// TIA Portal project "TIA_ControlTankSystem_VCSimit" (V16)

(* hardware
DEVICE "S71500/ET200MP station_1"  S7-1500 station
   slot 0: "Rail_0"  Rack  6ES7 590-1***0-0AA0
   slot 1: "PLC_1"  CPU 1511-1 PN  6ES7 511-1AK01-0AB0  V2.6
      slot 3: "CPU display_1"  6ES7591-1AA00-0AA0
      slot 32768: "PROFINET interface_1"  X1
         slot 32769: "Port_1"  X1 P1
         slot 32770: "Port_2"  X1 P2
DEVICE "S71500/ET200MP station_2"  S7-1500 station
   slot 0: "Rail_0"  Rack  6ES7 590-1***0-0AA0
   slot 1: "PLC_2"  CPU 1511-1 PN  6ES7 511-1AK01-0AB0  V2.8
      slot 3: "CPU display_1"  6ES7591-1AA00-0AA0
      slot 32768: "PROFINET interface_1"  X1
         slot 32769: "Port_1"  X1 P1
         slot 32770: "Port_2"  X1 P2
      slot 34817: "Virtual CP interface port_1"  Virtual CP interface port  Virtual CP interface port
DEVICE "ET 200SP station_1"  ET 200SP-Station
   slot 0: "Rack_0"  Rack  6ES5 710-8MAx1
   slot 0: "IO device_1"  IM 155-6 PN HF  6ES7 155-6AU00-0CN0  V4.2
   slot 1: "DI 8x24VDC HF_1"  DI 8x24VDC HF  6ES7 131-6BF00-0CA0  V2.0
      slot 1: "DI 8x24VDC HF_1"  DI 8x24VDC HF
   slot 2: "DI 8x24VDC HF_2"  DI 8x24VDC HF  6ES7 131-6BF00-0CA0  V2.0
      slot 1: "DI 8x24VDC HF_2"  DI 8x24VDC HF
   slot 3: "DI 8x24VDC HF_3"  DI 8x24VDC HF  6ES7 131-6BF00-0CA0  V2.0
      slot 1: "DI 8x24VDC HF_3"  DI 8x24VDC HF
   slot 4: "DQ 8x24VDC/0.5A HF_1"  DQ 8x24VDC/0.5A HF  6ES7 132-6BF00-0CA0  V2.0
      slot 1: "DQ 8x24VDC/0.5A HF_1"  DQ 8x24VDC/0.5A HF
   slot 5: "DQ 8x24VDC/0.5A HF_2"  DQ 8x24VDC/0.5A HF  6ES7 132-6BF00-0CA0  V2.0
      slot 1: "DQ 8x24VDC/0.5A HF_2"  DQ 8x24VDC/0.5A HF
   slot 6: "AI 2xU/I 2-,4-wire HS_1"  AI 2xU/I 2-,4-wire HS  6ES7 134-6HB00-0DA1  V2.0
      slot 1: "AI 2xU/I 2-,4-wire HS_1"  AI 2xU/I 2-,4-wire HS
   slot 7: "AI 2xU/I 2-,4-wire HS_2"  AI 2xU/I 2-,4-wire HS  6ES7 134-6HB00-0DA1  V2.0
      slot 1: "AI 2xU/I 2-,4-wire HS_2"  AI 2xU/I 2-,4-wire HS
   slot 8: "AI 2xU/I 2-,4-wire HS_3"  AI 2xU/I 2-,4-wire HS  6ES7 134-6HB00-0DA1  V2.0
      slot 1: "AI 2xU/I 2-,4-wire HS_3"  AI 2xU/I 2-,4-wire HS
   slot 9: "AQ 2xU/I HS_1"  AQ 2xU/I HS  6ES7 135-6HB00-0DA1  V2.0
      slot 1: "AQ 2xU/I HS_1"  AQ 2xU/I HS
   slot 10: "AQ 2xU/I HS_2"  AQ 2xU/I HS  6ES7 135-6HB00-0DA1  V2.0
      slot 1: "AQ 2xU/I HS_2"  AQ 2xU/I HS
   slot 11: "Server module_1"  Server module  6ES7 193-6PA00-0AA0  V1.1
      slot 1: "Server module_1"  Server module
   slot 127: "BA 2xRJ45"  BA 2xRJ45  6ES7 193-6AR00-0AA0  V0.0
      slot 1: "Port_1"  X1 P1 R  6ES7 193-6AR00-0AA0  V0.0
      slot 2: "Port_2"  X1 P2 R  6ES7 193-6AR00-0AA0  V0.0
DEVICE "PC-System_1"  SIMATIC PC station
   slot 0: "SIMATIC PC station"  Rail  SIMATIC PC-Station  V1.0
      slot 125: "Stationmanager"  Station_Manager  V6.0.4
   slot 1: "HMI_RT_1"  WinCC RT Advanced  6AV2 104-0xxxx-xxxx  16.0.0.0
      slot 33792: "Computer interface"  Host interface
   slot 2: "IE general_1"  IE General  IE_CP  V8.2.0
*)

// ===== PLC "PLC_1"  CPU 1511-1 PN =====

VAR_GLOBAL   // PLC tag table "Default tag table"
   "Motor2_SpeedRaw" AT %MW0 : Int;
   "Motor2_Speed" AT %MD2 : Real;
   "Tank2_Level" AT %MD6 : Real;
   "Tank2_LevelRaw" AT %MW10 : Int;
   "Motor2_SpeedSPRaw" AT %MW12 : Int;
   "Motor2_SpeedSP" AT %MD14 : Real;
   "Motor2_VFDCMD" AT %M18.0 : Bool;
END_VAR

DATA_BLOCK "ReadBuffer"   // DB2
{ S7_Optimized_Access := 'FALSE' }
VERSION : 0.1
   VAR
      Speed_2 : Int;
      BoolStatus_2 : Word;
      Level_2 : Int;
   END_VAR
BEGIN
END_DATA_BLOCK

DATA_BLOCK "ModbusConfig"   // DB3
{ S7_Optimized_Access := 'TRUE' }
VERSION : 0.1
   VAR
      ReadConfig : TCON_IP_v4;
      WriteConfig : TCON_IP_v4;
   END_VAR
BEGIN
   ReadConfig.InterfaceId := 64;
   ReadConfig.ID := 30;
   ReadConfig.ActiveEstablished := true;
   ReadConfig.RemoteAddress.ADDR[1] := 192;
   ReadConfig.RemoteAddress.ADDR[2] := 168;
   ReadConfig.RemoteAddress.ADDR[3] := 0;
   ReadConfig.RemoteAddress.ADDR[4] := 12;
   ReadConfig.RemotePort := 502;
   ReadConfig.ConnectionType := 11;
   WriteConfig.InterfaceId := 64;
   WriteConfig.ID := 31;
   WriteConfig.ConnectionType := 11;
   WriteConfig.ActiveEstablished := true;
   WriteConfig.RemoteAddress.ADDR[1] := 192;
   WriteConfig.RemoteAddress.ADDR[2] := 168;
   WriteConfig.RemoteAddress.ADDR[3] := 0;
   WriteConfig.RemoteAddress.ADDR[4] := 12;
   WriteConfig.RemotePort := 502;
END_DATA_BLOCK

DATA_BLOCK "WriteBuffer"   // DB4
{ S7_Optimized_Access := 'FALSE' }
VERSION : 0.1
   VAR
      SpeedSP_2 : Int;
      BoolStatus_2 : Int;
   END_VAR
BEGIN
END_DATA_BLOCK

DATA_BLOCK "Motor2"   // DB5
{ S7_Optimized_Access := 'FALSE' }
VERSION : 0.1
   VAR
      Speed : Real;
      SpeedSP : Real;
      Status : Bool;
      Fault : Bool;
      Start : Bool;
      Stop : Bool;
   END_VAR
BEGIN
END_DATA_BLOCK

DATA_BLOCK "Tank2"   // DB6
{ S7_Optimized_Access := 'FALSE' }
VERSION : 0.1
   VAR
      Level : Real;
      LevelSP : Real;
      AlarmLow : Bool;
      AlarmHigh : Bool;
      PIDST : Bool;
   END_VAR
BEGIN
END_DATA_BLOCK

ORGANIZATION_BLOCK "Main"   // OB1, LAD, ProgramCycle
TITLE = "Main Program Sweep (Cycle)"
{ S7_Optimized_Access := 'TRUE' }
VERSION : 0.1
   VAR_INPUT
      Initial_Call : Bool;   // Initial call of this OB
      Remanence : Bool;   // =True, if remanent data are available
   END_VAR
BEGIN
END_ORGANIZATION_BLOCK

ORGANIZATION_BLOCK "ModbusClient"   // OB123, LAD, ProgramCycle
TITLE = "Main Program Sweep (Cycle)"
{ S7_Optimized_Access := 'TRUE' }
VERSION : 0.1
   VAR_INPUT
      Initial_Call : Bool;   // Initial call of this OB
      Remanence : Bool;   // =True, if remanent data are available
   END_VAR
BEGIN

REGION Network 1
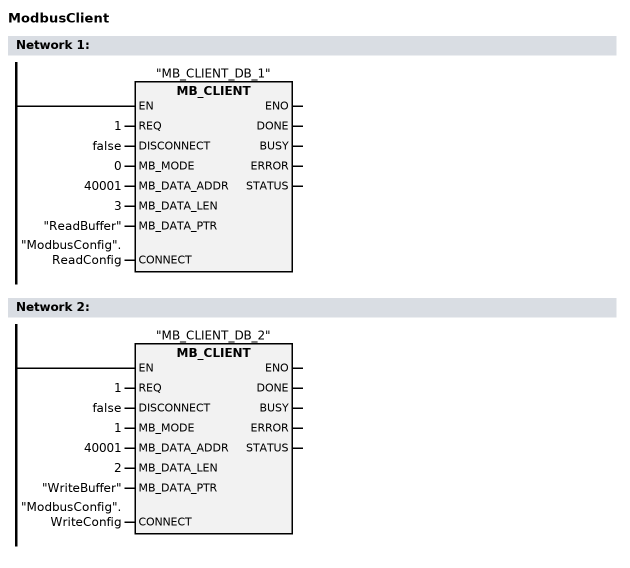
   "MB_CLIENT_DB_1"(REQ := 1,   // MB_CLIENT
                    DISCONNECT := false,
                    MB_MODE := 0,
                    MB_DATA_ADDR := 40001,
                    MB_DATA_LEN := 3,
                    MB_DATA_PTR := "ReadBuffer",
                    CONNECT := "ModbusConfig".ReadConfig);
END_REGION

REGION Network 2
   "MB_CLIENT_DB_2"(REQ := 1,   // MB_CLIENT
                    DISCONNECT := false,
                    MB_MODE := 1,
                    MB_DATA_ADDR := 40001,
                    MB_DATA_LEN := 2,
                    MB_DATA_PTR := "WriteBuffer",
                    CONNECT := "ModbusConfig".WriteConfig);
END_REGION
END_ORGANIZATION_BLOCK

ORGANIZATION_BLOCK "ModbusClientMapping"   // OB124, SCL, ProgramCycle
TITLE = "Main Program Sweep (Cycle)"
{ S7_Optimized_Access := 'TRUE' }
VERSION : 0.1
   VAR_INPUT
      Initial_Call : Bool;   // Initial call of this OB
      Remanence : Bool;   // =True, if remanent data are available
   END_VAR
BEGIN
   "Motor2".Status := "ReadBuffer".BoolStatus_2.%X0;
   "Motor2".Fault := "ReadBuffer".BoolStatus_2.%X1;
   "Motor2".Start := "ReadBuffer".BoolStatus_2.%X2;
   "Motor2".Stop := "ReadBuffer".BoolStatus_2.%X3;

   "Motor2_SpeedRaw" := "ReadBuffer".Speed_2;
   "Tank2_LevelRaw" := "ReadBuffer".Level_2;

   "WriteBuffer".SpeedSP_2 := "Motor2_SpeedSPRaw";
   "WriteBuffer".BoolStatus_2.%X0 := "Tank2".AlarmLow;
   "WriteBuffer".BoolStatus_2.%X1 := "Tank2".AlarmHigh;
   "WriteBuffer".BoolStatus_2.%X2 := "Motor2_VFDCMD";
END_ORGANIZATION_BLOCK

// ===== PLC "PLC_2"  CPU 1511-1 PN =====

VAR_GLOBAL   // PLC tag table "Default tag table"
   "SpeedRaw" AT %MW0 : Word;
   "LevelRaw" AT %MW2 : Word;
   "SpeedSP" AT %MW4 : Word;
   "Status" AT %M6.0 : Bool;
   "Fault" AT %M6.1 : Bool;
   "Start" AT %M6.2 : Bool;
   "Stop" AT %M6.3 : Bool;
   "AlarmLow" AT %M6.4 : Bool;
   "AlarmHigh" AT %M6.5 : Bool;
   "TS2_Status" AT %I0.0 : Bool;
   "TS2_Fault" AT %I0.1 : Bool;
   "TS2_Start" AT %I0.2 : Bool;
   "TS2_Stop" AT %I0.3 : Bool;
   "TS2_VFDCMD" AT %Q0.0 : Bool;
   "TS2_AlarmLow" AT %Q0.1 : Bool;
   "TS2_AlarmHigh" AT %Q0.2 : Bool;
   "TS2_Speed" AT %IW3 : Int;
   "TS2_Level" AT %IW5 : Int;
   "TS2_SpeedSP" AT %QW2 : Int;
END_VAR

DATA_BLOCK "ReadBuffer"   // DB2
{ S7_Optimized_Access := 'FALSE' }
VERSION : 0.1
   VAR
      Speed_2 : Int := 27648;
      BoolStatus_2 : Word;
      Level_2 : Int;
   END_VAR
BEGIN
END_DATA_BLOCK

DATA_BLOCK "ModbusConfig"   // DB3
{ S7_Optimized_Access := 'TRUE' }
VERSION : 0.1
   VAR
      ReadConfig : TCON_IP_v4;
      WriteConfig : TCON_IP_v4;
   END_VAR
BEGIN
   ReadConfig.InterfaceId := 64;
   ReadConfig.ID := 30;
   ReadConfig.ActiveEstablished := false;
   ReadConfig.RemoteAddress.ADDR[1] := 192;
   ReadConfig.RemoteAddress.ADDR[2] := 168;
   ReadConfig.RemoteAddress.ADDR[3] := 0;
   ReadConfig.RemoteAddress.ADDR[4] := 11;
   ReadConfig.RemotePort := 0;
   ReadConfig.ConnectionType := 11;
   WriteConfig.InterfaceId := 64;
   WriteConfig.ID := 31;
   WriteConfig.ConnectionType := 11;
   WriteConfig.ActiveEstablished := false;
   WriteConfig.RemoteAddress.ADDR[1] := 192;
   WriteConfig.RemoteAddress.ADDR[2] := 168;
   WriteConfig.RemoteAddress.ADDR[3] := 0;
   WriteConfig.RemoteAddress.ADDR[4] := 11;
   WriteConfig.RemotePort := 0;
   ReadConfig.LocalPort := 502;
   WriteConfig.LocalPort := 502;
END_DATA_BLOCK

DATA_BLOCK "WriteBuffer"   // DB4
{ S7_Optimized_Access := 'FALSE' }
VERSION : 0.1
   VAR
      SpeedSP_2 : Int;
      BoolStatus_2 : Int;
   END_VAR
BEGIN
END_DATA_BLOCK

ORGANIZATION_BLOCK "Main"   // OB1, LAD, ProgramCycle
TITLE = "Main Program Sweep (Cycle)"
{ S7_Optimized_Access := 'TRUE' }
VERSION : 0.1
   VAR_INPUT
      Initial_Call : Bool;   // Initial call of this OB
      Remanence : Bool;   // =True, if remanent data are available
   END_VAR
BEGIN
END_ORGANIZATION_BLOCK

ORGANIZATION_BLOCK "ModbusServer"   // OB123, LAD, ProgramCycle
TITLE = "Main Program Sweep (Cycle)"
{ S7_Optimized_Access := 'TRUE' }
VERSION : 0.1
   VAR_INPUT
      Initial_Call : Bool;   // Initial call of this OB
      Remanence : Bool;   // =True, if remanent data are available
   END_VAR
BEGIN

REGION Network 1
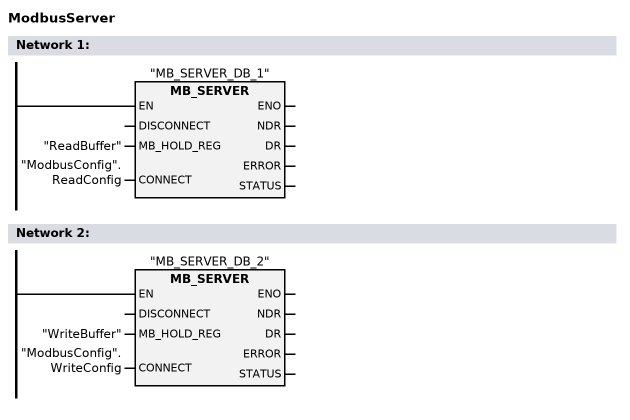
   "MB_SERVER_DB_1"(MB_HOLD_REG := "ReadBuffer", CONNECT := "ModbusConfig".ReadConfig);   // MB_SERVER
END_REGION

REGION Network 2
   "MB_SERVER_DB_2"(MB_HOLD_REG := "WriteBuffer", CONNECT := "ModbusConfig".WriteConfig);   // MB_SERVER
END_REGION
END_ORGANIZATION_BLOCK

ORGANIZATION_BLOCK "ModbusServerMapping"   // OB124, SCL, ProgramCycle
TITLE = "Main Program Sweep (Cycle)"
{ S7_Optimized_Access := 'TRUE' }
VERSION : 0.1
   VAR_INPUT
      Initial_Call : Bool;   // Initial call of this OB
      Remanence : Bool;   // =True, if remanent data are available
   END_VAR
BEGIN
   "ReadBuffer".Speed_2 := "TS2_Speed";
   "ReadBuffer".Level_2 := "TS2_Level";
   "ReadBuffer".BoolStatus_2.%X0 := "TS2_Status";
   "ReadBuffer".BoolStatus_2.%X1 := "TS2_Fault";
   "ReadBuffer".BoolStatus_2.%X2 := "TS2_Start";
   "ReadBuffer".BoolStatus_2.%X3 := "TS2_Stop";

   "TS2_SpeedSP" := "WriteBuffer".SpeedSP_2;
   "TS2_AlarmLow" := "WriteBuffer".BoolStatus_2.%X0;
   "TS2_AlarmHigh" := "WriteBuffer".BoolStatus_2.%X1;
   "TS2_VFDCMD" := "WriteBuffer".BoolStatus_2.%X2;
END_ORGANIZATION_BLOCK

(* ===== HMI "HMI_RT_1" =====
system functions are stored by id; their names below are inferred from use
connection "HMI_Connection_1": ETHERNET, S7_1500_OMS

HMI tags "Default tag table"
   "Motor2_SpeedRaw" : Int = PLC Motor2_SpeedRaw AT %MW0, 1 s
   "Tank2_LevelRaw" : Int = PLC Tank2_LevelRaw AT %MW10, 1 s

screen "Screen_1" 1024x768
   IOField "I/O field_1" at 94,105 size 96x32; FormatPattern s99999
      ProcessValue <- "Motor2_SpeedRaw"
   TextField "Text field_1" at 91,72 size 150x22; Text 'Motor 2 Raw Speed'
   IOField "I/O field_2" at 290,109 size 96x32; FormatPattern s99999
      ProcessValue <- "Tank2_LevelRaw"
   TextField "Text field_2" at 281,72 size 137x22; Text 'Tank 2 Raw Level'
   Button "Button_1" at 290,301 size 96x32; TextOff 'Exit'
      on Click: StopRuntime(0)
*)